// HW status for XYZ axis
TYPE ST_HW_STATUS_XYZ :
STRUCT
	bEStopOK:BOOL;
	fStepperTemp: LREAL;
	bLimitMax:BOOL;
	bLimitMin:BOOL;
	bLimitMaxMax:BOOL;
	bLimitMinMin:BOOL;
	bSumILOK:BOOL;
	bManualInterlockOverride:BOOL;
	bHwStatusOK:BOOL;  // Staatus of hardware (IPOS, EL7201, EL3214..)
	
	//Only X and Y
	bBrakeReleased: BOOL;
	
	//Only for Z
    bLimitMinPark:BOOL;
	bLimitMinMinPark:BOOL;	
	bParkingRangeEnabled:BOOL;
END_STRUCT
END_TYPE

(* stored: Version 1.1.0.1, ProductVersion 3.1.4024.6
   DUT ST_HW_STATUS_XYZ: Id {0c896078-d474-44e5-911d-70505f51c1b8} *)
